// TwinCAT 3 PLC project AccelerationSensor
// ProgramVersion: 3.1.0.8
// libraries:
//   Tc2_SerialCom, * (Beckhoff Automation GmbH)
//   Tc2_Standard, * (Beckhoff Automation GmbH)
//   Tc2_Utilities, * (Beckhoff Automation GmbH)
//   Tc3_Module, * (Beckhoff Automation GmbH)
// project tree:
//   GVLs/ AccelerationSensor.TcGVL, ActivationStatus.TcDUT (not stored), DUT.TcDUT, GuidanceSystemSTM.TcDUT, GVL.TcGVL, HighLevelCondition.TcDUT (not stored), HLSInputData.TcDUT, HLSInputData_1.TcDUT, HLSInputs.TcDUT, HLSOutputs.TcDUT, LEDColor.TcDUT (not stored), LEDMode.TcDUT, LevitationSystemSTM.TcDUT, OperationControlCommands.TcDUT, ServiceModuleSTM.TcDUT, SubLevelCondition.TcDUT (not stored), TopLevelSTM.TcDUT
//   / PlcTask_Fast.TcTTO, PlcTask_Standard.TcTTO (not stored)
//   POUs/ FB_AccelerationSensor.TcPOU, FB_SerialComRS232.TcPOU, ITF_HighLevelSystem.TcIO, ITF_SubSystem.TcIO, MAIN.TcPOU
//   POUs/Mit Background/ Background.TcPOU (not stored), BackgroundEL.TcPOU, FB_SerialCom.TcPOU
// real-time tasks:
//   TASK PlcTask_Fast: cycle T#1ms, priority 19, ADS port 350
//   TASK PlcTask_Standard: cycle T#1ms, priority 20, ADS port 351
// I/O:
//   DEVICE Gerät 1 (EtherCAT), AmsNetId 10.183.66.136.2.1
//     Klemme 1 (EK1100) [EK1100 EtherCAT-Koppler (2A E-Bus)]
//       Klemme 2 (EL6001) [EL6001 Schnittstelle (RS232)]
//       Klemme 3 (EL9011) [EL9011 Endklemme]
// variable links:
//   AccelerationSensor/AccelerationSensor Instance <-> Device 1 (EtherCAT)/Term 1 (EK1100)/Term 2 (EL6001)
//     PlcTask_Standard Inputs/AccelerationSensor.stEL6001In @bit {16..184 step 8} <-> COM Inputs/Data In {0..21}  (22 links)
//     PlcTask_Standard Inputs/AccelerationSensor.stEL6001In <-> COM Inputs/Status
//     PlcTask_Standard Outputs/AccelerationSensor.stEL6001Out <-> COM Outputs/Ctrl
//     PlcTask_Standard Outputs/AccelerationSensor.stEL6001Out @bit {16..184 step 8} <-> COM Outputs/Data Out {0..21}  (22 links)

CONFIGURATION AccelerationSensor
    RESOURCE PLC ON TwinCAT3
        TASK PlcTask_Fast(INTERVAL := T#1ms, PRIORITY := 19);
        PROGRAM Background WITH PlcTask_Fast : Background;
    END_RESOURCE
END_CONFIGURATION

// ---- GVLs/DUT.TcDUT
TYPE DUT :
STRUCT
	b : BOOL;
	n : BOOL;
	m : BOOL;
END_STRUCT
END_TYPE

// ---- GVLs/GuidanceSystemSTM.TcDUT
{attribute 'qualified_only'}
{attribute 'strict'}
TYPE GuidanceSystemSTM :
(
	Idling,
	Initialising,
	PreRunning,
	Running,
	PostRunning
);
END_TYPE

// ---- GVLs/HLSInputData.TcDUT
TYPE HLSInputData :
STRUCT
	//In
	iIn : INT;
END_STRUCT
END_TYPE

// ---- GVLs/HLSInputData_1.TcDUT
TYPE HLSInputData_1 :
STRUCT
	//In
	iIn : INT;
	
	//Out
	iOut : INT;
END_STRUCT
END_TYPE

// ---- GVLs/HLSInputs.TcDUT
TYPE HLSInputs :
STRUCT
	iIn : INT;
END_STRUCT
END_TYPE

// ---- GVLs/HLSOutputs.TcDUT
TYPE HLSOutputs :
STRUCT
	iOut : INT;
END_STRUCT
END_TYPE

// ---- GVLs/LEDMode.TcDUT
{attribute 'qualified_only'}
{attribute 'strict'}
TYPE LEDMode :
(
	Off,
	On,
	Dimmed,
	SlowFlashing,
	FastFlashing
);
END_TYPE

// ---- GVLs/LevitationSystemSTM.TcDUT
{attribute 'qualified_only'}
{attribute 'strict'}
TYPE LevitationSystemSTM :
(
	Idling,
	Stationary,
	Transitioning,
	HoldingAirGap,
	TransitioningToZero
);
END_TYPE

// ---- GVLs/OperationControlCommands.TcDUT
TYPE OperationControlCommands :
STRUCT
	bStartOperational : BOOL;
	bStopOperational : BOOL;
	bGoToError : BOOL;
	bAckError : BOOL;
	nOperationMode : BYTE;
END_STRUCT
END_TYPE

// ---- GVLs/ServiceModuleSTM.TcDUT
{attribute 'qualified_only'}
{attribute 'strict'}
TYPE ServiceModuleSTM :
(
	Idling,
	Waiting,
	Running,
	PostRunning,
	PreparingForError
);
END_TYPE

// ---- GVLs/TopLevelSTM.TcDUT
{attribute 'qualified_only'}
{attribute 'strict'}
TYPE TopLevelSTM :
(
	STARTUP,
	READY,
	OPERATIONAL,
	SHUTDOWN,
	ERROR
)USINT;
END_TYPE

// ---- GVLs/AccelerationSensor.TcGVL
VAR_GLOBAL
	stEL6001In AT %I*	: EL6inData22B;		//**To EL6021 Inputs**
	stEL6001Out AT %Q*	: EL6outData22B;	//**To EL6021 Outputs**
END_VAR

// ---- GVLs/GVL.TcGVL
VAR_GLOBAL
	RxBufferEL			: ComBuffer;	(* Receive data buffer; used with all receive function blocks *)
	TxBufferEL			: ComBuffer;	(* Transmit data buffer; used with all receive function blocks *)
END_VAR

// ---- POUs/ITF_HighLevelSystem.TcIO
INTERFACE ITF_HighLevelSystem

PROPERTY eActivationStatus : ActivationStatus
GET
END_GET
SET
END_SET
END_PROPERTY

PROPERTY PUBLIC eCondition : HighLevelCondition
GET
END_GET
END_PROPERTY

PROPERTY PUBLIC nErrorID : UDINT
GET
END_GET
END_PROPERTY

END_INTERFACE

// ---- POUs/ITF_SubSystem.TcIO
INTERFACE ITF_SubSystem

PROPERTY PUBLIC eCondition : SubLevelCondition
GET
END_GET
END_PROPERTY

PROPERTY PUBLIC nErrorID : UDINT
GET
END_GET
END_PROPERTY

END_INTERFACE

// ---- POUs/FB_AccelerationSensor.TcPOU
FUNCTION_BLOCK FB_AccelerationSensor IMPLEMENTS ITF_SubSystem
VAR_OUTPUT
	aAccelerationValues : ARRAY [0..2] OF REAL;
END_VAR
VAR
	//Local
	fbEL6001	: FB_SerialComRS232;
	fPacketRate : REAL := 0;
	bStartPacketCount : BOOL;
	
	fbTimer : TON;
	fbReset : TON;
	fbTrigger : R_TRIG;
	nCounter1 : UDINT;
	nCounter2 : UDINT;
	aPackets : ARRAY [0..9] OF UDINT;
	i : UDINT := 0;
	nSum : UDINT := 0;
	bTrigger : BOOL := FALSE;
	
	//ErrorBits
	bCommunicationError : BIT;
	bOutOfRange : BIT;
END_VAR
VAR CONSTANT
	fGravitationalAcceleration : REAL := 9.81;  					//in m/s^2
END_VAR

fbEL6001(stEL6001In:=AccelerationSensor.stEL6001In, stEL6001Out:=AccelerationSensor.stEL6001Out);

aAccelerationValues := fbEL6001.aAcceleration;

doPacketCount();

METHOD PRIVATE doCheckRange : BOOL
VAR_INPUT
	aValues : ARRAY [0..2] OF REAL;
	fMax : REAL;
END_VAR
IF ABS(aValues[0]) <= fMax AND ABS(aValues[1]) <= fMax AND ABS(aValues[2]) <= fMax THEN
	doCheckRange := TRUE;
ELSE
	doCheckRange := FALSE;
END_IF
END_METHOD

METHOD PRIVATE doPacketCount
VAR_INPUT
END_VAR
fbTimer(IN := bStartPacketCount, PT := T#1S);
fbTrigger(CLK := fbTimer.IN);

IF fbTrigger.Q THEN
	nCounter1 := fbEL6001.nReceiveCounter;
END_IF

IF fbTimer.Q THEN
	nCounter2 := fbEL6001.nReceiveCounter;
	aPackets[i] := nCounter2 - nCounter1;
	nSum := nSum + aPackets[i];
	i := i + 1;
	bTrigger := TRUE;
	bStartPacketCount := FALSE;
END_IF

IF i = 10 THEN
	bTrigger := FALSE;
	fPacketRate := (UDINT_TO_REAL(nSum) / UDINT_TO_REAL(i));
	i := 0;
	nSum := 0;
END_IF

fbReset(IN := bTrigger, PT := T#3S);
IF fbReset.Q THEN
	bStartPacketCount := TRUE;
	bTrigger := FALSE;
END_IF
END_METHOD

PROPERTY PUBLIC eCondition : SubLevelCondition
GET
IF nErrorID <> 0 THEN
	eCondition := SubLevelCondition.ERROR;
ELSE
	eCondition := SubLevelCondition.RUN;
END_IF
END_GET
END_PROPERTY

PROPERTY PUBLIC nErrorID : UDINT
GET
IF fbEL6001.eReceiveErrorID <> COMERROR_NOERROR THEN
	bCommunicationError := TRUE;
ELSE
	bCommunicationError := FALSE;
END_IF

bOutOfRange := NOT doCheckRange(aValues:=aAccelerationValues, fMax:=2*fGravitationalAcceleration);


nErrorID.0 := bCommunicationError;
nErrorID.1 := bOutOfRange;
END_GET
END_PROPERTY

END_FUNCTION_BLOCK

// ---- POUs/FB_SerialComRS232.TcPOU
FUNCTION_BLOCK FB_SerialComRS232
VAR_IN_OUT

	stEL6001In : EL6inData22B;
	stEL6001Out : EL6outData22B;
END_VAR
VAR_OUTPUT
	aAcceleration : ARRAY [0..2] OF REAL;
	eReceiveErrorID	: ComError_t;
	nReceiveCounter	: UDINT;
END_VAR
VAR

	//Receive Buffer
	fbEL6001Ctrl		: SerialLineControl;
	TxBuffer	: ComBuffer;
	RxBuffer	: ComBuffer;
	//Receive Data
	fbReceive		: ReceiveData;
	nPrefix : ARRAY[0..1] OF BYTE;
	aReceiveData : ARRAY [0..15] OF BYTE;
	nPacketID : BYTE := 37;
	nPacketLength : BYTE := 12;	
	
	nCRC : WORD;
	nCheckCRC : WORD;
	nPointerCRC : POINTER TO WORD;
	aCRC : ARRAY [0..1] OF BYTE;	
	aDataArray : ARRAY[0..11] OF BYTE;
	i : USINT;
	aAccX : ARRAY [0..3] OF BYTE;
	aAccY : ARRAY [0..3] OF BYTE;
	aAccZ : ARRAY [0..3] OF BYTE;
	fPointerToX : POINTER TO REAL;
    fAccX : REAL;
	fPointerToY : POINTER TO REAL;
    fAccY : REAL;
	fPointerToZ : POINTER TO REAL;
    fAccZ : REAL;
END_VAR

fbEL6001Ctrl(
	Mode:= SERIALLINEMODE_EL6_22B, 
	pComIn:= ADR(stEL6001In), 
	pComOut:= ADR(stEL6001Out), 
	SizeComIn:= SIZEOF(stEL6001In), 
	Error=> , 
	ErrorID=> , 
	TxBuffer:= TxBuffer, 
	RxBuffer:= RxBuffer);

nPrefix[0] := nPacketID;
nPrefix[1] := nPacketLength;

fbReceive(
	RXbuffer:= RxBuffer,
	pPrefix := ADR(nPrefix),
	LenPrefix := 2,
	pReceiveData := ADR(aReceiveData),
	SizeReceiveData  := 16,								
	Error => eReceiveErrorID,
	DataReceived=>);
		
IF fbReceive.DataReceived THEN							
	nReceiveCounter := nReceiveCounter + 1;
END_IF

doCRC16Check();
doCalculateAccValues();

METHOD PRIVATE doCalculateAccValues
VAR_INPUT
END_VAR
IF nCheckCRC = nCRC THEN
	aAccX[0] := aReceiveData[4];
	aAccX[1] := aReceiveData[5];
	aAccX[2] := aReceiveData[6];
	aAccX[3] := aReceiveData[7];
	fPointerToX := ADR(aAccX);
	fAccX := fPointerToX^;
	
	aAccY[0] := aReceiveData[8];
	aAccY[1] := aReceiveData[9];
	aAccY[2] := aReceiveData[10];
	aAccY[3] := aReceiveData[11];
	fPointerToY := ADR(aAccY);
	fAccY := fPointerToY^;
	
	aAccZ[0] := aReceiveData[12];
	aAccZ[1] := aReceiveData[13];
	aAccZ[2] := aReceiveData[14];
	aAccZ[3] := aReceiveData[15];
	fPointerToZ := ADR(aAccZ);
	fAccZ := fPointerToZ^;
END_IF

aAcceleration[0] := fAccX;
aAcceleration[1] := fAccY;
aAcceleration[2] := fAccZ;
END_METHOD

METHOD PRIVATE doCRC16Check : BOOL
VAR_INPUT
END_VAR
FOR i:=0 TO 11 DO
	aDataArray[i] := aReceiveData[i+4];
END_FOR


nCRC := F_DATA_TO_CRC16_CCITT(
	pData := ADR(aDataArray),
	cbData := BYTE_TO_UDINT(nPacketLength),
	crc := 16#FFFF);

aCRC[0] := aReceiveData[2];
aCRC[1] := aReceiveData[3];
nPointerCRC := ADR(aCRC);
nCheckCRC := nPointerCRC^;
END_METHOD

END_FUNCTION_BLOCK

// ---- POUs/MAIN.TcPOU
PROGRAM MAIN
VAR
	fbIMU : FB_AccelerationSensor;
	
	x : REAL;
	y : REAL;
	z : REAL;
	
	acc : ARRAY [0..2] OF REAL;

//	fbEL6001	: FB_SerialCom;
	
//	(* exchange buffers with background communication with the PC COM port device *)
//	RxBufferPcCom	: ComBuffer;	(* Receive data buffer; used with all receive function blocks *)
//	TxBufferPcCom	: ComBuffer;	(* Transmit data buffer; used with all receive function blocks *)
	
//	acc_x : REAL;
//	acc_y : REAL;	
//	acc_z : REAL;
////	acc_x2 : REAL;
////	acc_y2 : REAL;	
////	acc_z2 : REAL;
////	acc_x3 : REAL;
////	acc_y3 : REAL;	
////	acc_z3 : REAL;
////	acc_x4 : REAL;
////	acc_y4 : REAL;	
////	acc_z4 : REAL;

//	fbTimer : TON;
//	fbReset : TON;
//	fbTrigger : R_TRIG;
//	iCounter1 : UDINT;
//	iCounter2 : UDINT;
//	a_iPackets : ARRAY [0..9] OF UDINT;
//	i : UDINT := 0;
//	iSum : UDINT := 0;
//	rPacketRate : REAL := 0;
//	bTrigger : BOOL := FALSE;
//	bCount : BOOL;

END_VAR

fbIMU();

acc := fbIMU.aAccelerationValues;

x := acc[0];
y := acc[1];
z := acc[2];



//fbEL6001(TxBuffer:=TxBufferEL, RxBuffer:=RxBufferEL);

//acc_x := fbEL6001.getAccelerationValueX;
//acc_y := fbEL6001.getAccelerationValueY;
//acc_z := fbEL6001.getAccelerationValueZ;

//acc_x2 := fbEL6001.getAccelerationValueX2;
//acc_y2 := fbEL6001.getAccelerationValueY2;
//acc_z2 := fbEL6001.getAccelerationValueZ2;

//acc_x3 := fbEL6001.getAccelerationValueX3;
//acc_y3 := fbEL6001.getAccelerationValueY3;
//acc_z3 := fbEL6001.getAccelerationValueZ3;

//acc_x4 := fbEL6001.getAccelerationValueX4;
//acc_y4 := fbEL6001.getAccelerationValueY4;
//acc_z4 := fbEL6001.getAccelerationValueZ4;

doPacketCount();					//start packet count by setting bCount 'true' --> rPacketRate shows average rate per second

METHOD doPacketCount : REAL
VAR_INPUT
END_VAR
//fbTimer(IN := bCount, PT := T#1S);
//fbTrigger(CLK := fbTimer.IN);

//IF fbTrigger.Q THEN
//	iCounter1 := fbEL6001.nReceiveCounter;
//END_IF

//IF fbTimer.Q THEN
//	iCounter2 := fbEL6001.nReceiveCounter;
//	a_iPackets[i] := iCounter2 - iCounter1;
//	iSum := iSum + a_iPackets[i];
//	i := i + 1;
//	bTrigger := TRUE;
//	bCount := FALSE;
//END_IF

//IF i = 10 THEN
//	bTrigger := FALSE;
//	rPacketRate := (UDINT_TO_REAL(iSum) / UDINT_TO_REAL(i));			//times amount of packets
//	i := 0;
//	iSum := 0;
//END_IF

//fbReset(IN := bTrigger, PT := T#3S);
//IF fbReset.Q THEN
//	bCount := TRUE;
//	bTrigger := FALSE;
//END_IF
END_METHOD

END_PROGRAM

// ---- POUs/Mit Background/BackgroundEL.TcPOU
PROGRAM BackgroundEL
VAR
	(* background communication with the EL6001 terminal *)
	fbEL6001Ctrl		: SerialLineControl;
	bEL6001CtrlError	: BOOL;
	eEL6001CtrlErrorID	: ComError_t;
	(* 	I/O variables for a EL6001 terminal*)
	stIn_EL6001 AT %I*	: EL6inData22B;	(* linked to the EL6001 in the TwinCAT System Manager *)
	stOut_EL6001 AT %Q*	: EL6outData22B;(* linked to the EL6001 in the TwinCAT System Manager *)
END_VAR

fbEL6001Ctrl(
	Mode:= SERIALLINEMODE_EL6_22B, 
	pComIn:= ADR(stIn_EL6001), 
	pComOut:= ADR(stOut_EL6001), 
	SizeComIn:= SIZEOF(stIn_EL6001), 
	Error=> , 
	ErrorID=> , 
	TxBuffer:= TxBufferEL, 
	RxBuffer:= RxBufferEL );
IF fbEL6001Ctrl.Error THEN
	bEL6001CtrlError := TRUE;
	eEL6001CtrlErrorID := fbEL6001Ctrl.ErrorID;
END_IF

END_PROGRAM

// ---- POUs/Mit Background/FB_SerialCom.TcPOU
FUNCTION_BLOCK FB_SerialCom
VAR_IN_OUT
	TxBuffer	: ComBuffer;
	RxBuffer	: ComBuffer;
END_VAR
VAR
	fbReceive		: ReceiveData;
	eReceiveErrorID	: ComError_t;
	nReceiveCounter	: UDINT;
	prefix : ARRAY[0..1] OF BYTE;
	receivedata : ARRAY [0..15] OF BYTE;					//decrease or increase by 17 pro packet
	packet_ID : BYTE := 37;
	packet_length : BYTE := 12;	
	
	//First Package
	crc : WORD;
	crc_check : WORD;
	pt_crc : POINTER TO WORD;
	crc12 : ARRAY [0..1] OF BYTE;	
	dataArray : ARRAY[0..11] OF BYTE;
	i : USINT;
	acc_x : ARRAY [0..3] OF BYTE;
	acc_y : ARRAY [0..3] OF BYTE;
	acc_z : ARRAY [0..3] OF BYTE;
	pt_x : POINTER TO REAL;
    x_acc : REAL;
	pt_y : POINTER TO REAL;
    y_acc : REAL;
	pt_z : POINTER TO REAL;
    z_acc : REAL;
	

//	//Second Package
//	bSecondReceivedData: ARRAY [0..16] OF BYTE;
//	dataArray2 : ARRAY[0..11] OF BYTE;
//	crc2 : WORD;
//	crc122 : ARRAY [0..1]OF BYTE;
//	pt_crc2 : POINTER TO WORD;
//	crc_check2 : WORD;
//	k2 : USINT;
//	LRCsum2 : BYTE;
//	LRC2 : BYTE;
//	LRCchecked2 : BOOL;
//	j2 : USINT;
//	bIn2 : BOOL;
//	acc_x2 : ARRAY [0..3] OF BYTE;
//	acc_y2 : ARRAY [0..3] OF BYTE;
//	acc_z2 : ARRAY [0..3] OF BYTE;
//	pt_x2 : POINTER TO REAL;
//  x_acc2 : REAL;
//	pt_y2 : POINTER TO REAL;
//  y_acc2 : REAL;
//	pt_z2 : POINTER TO REAL;
//  z_acc2 : REAL;
	
//	//Third Package
//	bThirdReceivedData: ARRAY [0..16] OF BYTE;
//	dataArray3 : ARRAY[0..11] OF BYTE;
//	crc3 : WORD;
//	crc123 : ARRAY [0..1]OF BYTE;
//	pt_crc3 : POINTER TO WORD;
//	crc_check3 : WORD;
//	k3 : USINT;
//	LRCsum3 : BYTE;
//	LRC3 : BYTE;
//	LRCchecked3 : BOOL;
//	j3 : USINT;
//	bIn3 : BOOL;
//	acc_x3 : ARRAY [0..3] OF BYTE;
//	acc_y3 : ARRAY [0..3] OF BYTE;
//	acc_z3 : ARRAY [0..3] OF BYTE;
//	pt_x3 : POINTER TO REAL;
//  x_acc3 : REAL;
//	pt_y3 : POINTER TO REAL;
//  y_acc3 : REAL;
//	pt_z3 : POINTER TO REAL;
//  z_acc3 : REAL;
	
//	//Fourth Package
//	bFourthReceivedData: ARRAY [0..16] OF BYTE;
//	dataArray4 : ARRAY[0..11] OF BYTE;
//	crc4 : WORD;
//	crc124 : ARRAY [0..1]OF BYTE;
//	pt_crc4 : POINTER TO WORD;
//	crc_check4 : WORD;
//	k4 : USINT;
//	LRCsum4 : BYTE;
//	LRC4 : BYTE;
//	LRCchecked4 : BOOL;
//	j4 : USINT;
//	bIn4 : BOOL;
//	acc_x4 : ARRAY [0..3] OF BYTE;
//	acc_y4 : ARRAY [0..3] OF BYTE;
//	acc_z4 : ARRAY [0..3] OF BYTE;
//	pt_x4 : POINTER TO REAL;
//  x_acc4 : REAL;
//	pt_y4 : POINTER TO REAL;
//  y_acc4 : REAL;
//	pt_z4 : POINTER TO REAL;
//  z_acc4 : REAL;
END_VAR

prefix[0] := packet_ID;
prefix[1] := packet_length;

fbReceive(
	RXbuffer:= RxBuffer,
	pPrefix := ADR(prefix),
	LenPrefix := 2,
	pReceiveData := ADR(receivedata),
	SizeReceiveData  := 16,											//decrease or increase by 17 per packet
	Error=> ,
	DataReceived=>,
		);
IF fbReceive.Error <> COMERROR_NOERROR THEN
	eReceiveErrorID := fbReceive.Error;
END_IF
IF fbReceive.DataReceived THEN										//check bIn* variables as well for multiple packets
	nReceiveCounter := nReceiveCounter + 1;
END_IF

doCRC16Check1();

//IF receivedata[17] = 37 AND receivedata[18] = 12 THEN				//decrease or increase by 17 per packet
//	bIn2 := TRUE;	
//	FOR k2:=0 TO 16 DO
//		bSecondReceivedData[k] := receivedata[k+16];
//	END_FOR
	
//	doLRCCheck2();
//	doCRC16Check2();
//ELSE
//	bIn2 := FALSE;
//END_IF


//IF receivedata[34] = 37 AND receivedata[35] = 12 THEN				//decrease or increase by 17 per packet
//	bIn3 := TRUE;	
//	FOR k3:=0 TO 16 DO
//		bThirdReceivedData[k3] := receivedata[k3+16];
//	END_FOR
	
//	doLRCCheck3();
//	doCRC16Check3();
//ELSE
//	bIn3 := FALSE;
//END_IF


//IF receivedata[51] = 37 AND receivedata[52] = 12 THEN			//decrease or increase by 17 per packet
//	bIn4 := TRUE;	
//	FOR k4:=0 TO 16 DO
//		bFourthReceivedData[k4] := receivedata[k4+16];
//	END_FOR
	
//	doLRCCheck4();
//	doCRC16Check4();
//ELSE
//	bIn4 := FALSE;
//END_IF

METHOD doCRC16Check1 : BOOL
VAR_INPUT
END_VAR
FOR i:=0 TO 11 DO
	dataArray[i] := receivedata[i+4];
END_FOR


crc := F_DATA_TO_CRC16_CCITT(
	pData := ADR(dataArray),
	cbData := BYTE_TO_UDINT(packet_length),
	crc := 16#FFFF);

crc12[0] := receivedata[2];
crc12[1] := receivedata[3];
pt_crc := ADR(crc12);
crc_check := pt_crc^;
END_METHOD

METHOD doCRC16Check2 : BOOL
VAR_INPUT
END_VAR
//FOR j2:=0 TO 11 DO
//	dataArray2[j] := bSecondReceivedData[j+5];
//END_FOR
	
	
//crc2 := F_DATA_TO_CRC16_CCITT(
//	pData := ADR(dataArray2),
//	cbData := BYTE_TO_UDINT(packet_length),
//	crc := 16#FFFF);

//crc122[0] := bSecondReceivedData[3];
//crc122[1] := bSecondReceivedData[4];
//pt_crc2 := ADR(crc122);
//crc_check2 := pt_crc2^;
END_METHOD

METHOD doCRC16Check3 : BOOL
VAR_INPUT
END_VAR
//FOR j3:=0 TO 11 DO
//	dataArray3[j3] := bThirdReceivedData[j3+5];
//END_FOR
	
	
//crc3 := F_DATA_TO_CRC16_CCITT(
//	pData := ADR(dataArray3),
//	cbData := BYTE_TO_UDINT(packet_length),
//	crc := 16#FFFF);

//crc123[0] := bThirdReceivedData[3];
//crc123[1] := bThirdReceivedData[4];
//pt_crc3 := ADR(crc123);
//crc_check3 := pt_crc3^;
END_METHOD

METHOD doCRC16Check4 : BOOL
VAR_INPUT
END_VAR
//FOR j4:=0 TO 11 DO
//	dataArray4[j4] := bFourthReceivedData[j4+5];
//END_FOR
	
	
//crc4 := F_DATA_TO_CRC16_CCITT(
//	pData := ADR(dataArray4),
//	cbData := BYTE_TO_UDINT(packet_length),
//	crc := 16#FFFF);

//crc124[0] := bFourthReceivedData[3];
//crc124[1] := bFourthReceivedData[4];
//pt_crc4 := ADR(crc124);
//crc_check4 := pt_crc4^;
END_METHOD

METHOD doLRCCheck2 : BOOL
VAR_INPUT
END_VAR
//LRCsum2 := (bSecondReceivedData[1] + bSecondReceivedData[2] + bSecondReceivedData[3] + bSecondReceivedData[4]) XOR 255;
//LRC2 := bSecondReceivedData[0] - 1;
//LRCchecked2 := (LRCsum2 = LRC2);
END_METHOD

METHOD doLRCCheck3 : BOOL
VAR_INPUT
END_VAR
//LRCsum3 := (bThirdReceivedData[1] + bThirdReceivedData[2] + bThirdReceivedData[3] + bThirdReceivedData[4]) XOR 255;
//LRC3 := bThirdReceivedData[0] - 1;
//LRCchecked3 := (LRCsum3 = LRC3);
END_METHOD

METHOD doLRCCheck4 : BOOL
VAR_INPUT
END_VAR
//LRCsum4 := (bFourthReceivedData[1] + bFourthReceivedData[2] + bFourthReceivedData[3] + bFourthReceivedData[4]) XOR 255;
//LRC4 := bFourthReceivedData[0] - 1;
//LRCchecked4 := (LRCsum4 = LRC4);
END_METHOD

PROPERTY getAccelerationValueX : REAL
GET
IF crc_check = crc THEN

	acc_x[0] := receivedata[4];
	acc_x[1] := receivedata[5];
	acc_x[2] := receivedata[6];
	acc_x[3] := receivedata[7];
	pt_x := ADR(acc_x);
	x_acc := pt_x^;
END_IF

getAccelerationValueX := x_acc;
END_GET
END_PROPERTY

PROPERTY getAccelerationValueX2 : REAL
GET
//IF LRCsum = LRC AND crc2 = crc_check2 THEN
//	acc_x2[0] := bSecondReceivedData[5];
//	acc_x2[1] := bSecondReceivedData[6];
//	acc_x2[2] := bSecondReceivedData[7];
//	acc_x2[3] := bSecondReceivedData[8];
//	pt_x2 := ADR(acc_x2);
//	x_acc2 := pt_x2^;
//END_IF

//getAccelerationValueX2 := x_acc2;
END_GET
END_PROPERTY

PROPERTY getAccelerationValueX3 : REAL
GET
//IF LRCsum3 = LRC3 AND crc3 = crc_check3 THEN
//	acc_x3[0] := bThirdReceivedData[5];
//	acc_x3[1] := bThirdReceivedData[6];
//	acc_x3[2] := bThirdReceivedData[7];
//	acc_x3[3] := bThirdReceivedData[8];
//	pt_x3 := ADR(acc_x3);
//	x_acc3 := pt_x3^;
//END_IF

//getAccelerationValueX3 := x_acc3;
END_GET
END_PROPERTY

PROPERTY getAccelerationValueX4 : REAL
GET
//IF LRCsum4 = LRC4 AND crc4 = crc_check4 THEN
//	acc_x4[0] := bFourthReceivedData[5];
//	acc_x4[1] := bFourthReceivedData[6];
//	acc_x4[2] := bFourthReceivedData[7];
//	acc_x4[3] := bFourthReceivedData[8];
//	pt_x4 := ADR(acc_x4);
//	x_acc4 := pt_x4^;
//END_IF

//getAccelerationValueX4 := x_acc4;
END_GET
END_PROPERTY

PROPERTY getAccelerationValueY : REAL
GET
IF crc_check = crc THEN
	
	acc_y[0] := receivedata[8];
	acc_y[1] := receivedata[9];
	acc_y[2] := receivedata[10];
	acc_y[3] := receivedata[11];
	pt_y := ADR(acc_y);
	y_acc := pt_y^;

END_IF
getAccelerationValueY := y_acc;
END_GET
END_PROPERTY

PROPERTY getAccelerationValueY2 : REAL
GET
//IF LRCsum = LRC AND crc2 = crc_check2 THEN
//	acc_y2[0] := bSecondReceivedData[9];
//	acc_y2[1] := bSecondReceivedData[10];
//	acc_y2[2] := bSecondReceivedData[11];
//	acc_y2[3] := bSecondReceivedData[12];
//	pt_y2 := ADR(acc_y2);
//	y_acc2 := pt_y2^;
//END_IF

//getAccelerationValueY2 := y_acc2;
END_GET
END_PROPERTY

PROPERTY getAccelerationValueY3 : REAL
GET
//IF LRCsum3 = LRC3 AND crc3 = crc_check3 THEN
//	acc_y3[0] := bThirdReceivedData[9];
//	acc_y3[1] := bThirdReceivedData[10];
//	acc_y3[2] := bThirdReceivedData[11];
//	acc_y3[3] := bThirdReceivedData[12];
//	pt_y3 := ADR(acc_y3);
//	y_acc3 := pt_y3^;
//END_IF

//getAccelerationValueY3 := y_acc3;
END_GET
END_PROPERTY

PROPERTY getAccelerationValueY4 : REAL
GET
//IF LRCsum4 = LRC4 AND crc4 = crc_check4 THEN
//	acc_y4[0] := bFourthReceivedData[9];
//	acc_y4[1] := bFourthReceivedData[10];
//	acc_y4[2] := bFourthReceivedData[11];
//	acc_y4[3] := bFourthReceivedData[12];
//	pt_y4 := ADR(acc_y4);
//	y_acc4 := pt_y4^;
//END_IF

//getAccelerationValueY4 := y_acc4;
END_GET
END_PROPERTY

PROPERTY getAccelerationValueZ : REAL
GET
IF crc_check = crc THEN
	
	acc_z[0] := receivedata[12];
	acc_z[1] := receivedata[13];
	acc_z[2] := receivedata[14];
	acc_z[3] := receivedata[15];
	pt_z := ADR(acc_z);
	z_acc := pt_z^;
END_IF

getAccelerationValueZ := z_acc;
END_GET
END_PROPERTY

PROPERTY getAccelerationValueZ2 : REAL
GET
//IF LRCsum = LRC AND crc2 = crc_check2 THEN
//	acc_z2[0] := bSecondReceivedData[13];
//	acc_z2[1] := bSecondReceivedData[14];
//	acc_z2[2] := bSecondReceivedData[15];
//	acc_z2[3] := bSecondReceivedData[16];
//	pt_z2 := ADR(acc_z2);
//	z_acc2 := pt_z2^;
//END_IF

//getAccelerationValueZ2 := z_acc2;
END_GET
END_PROPERTY

PROPERTY getAccelerationValueZ3 : REAL
GET
//IF LRCsum3 = LRC3 AND crc3 = crc_check3 THEN
//	acc_z3[0] := bThirdReceivedData[13];
//	acc_z3[1] := bThirdReceivedData[14];
//	acc_z3[2] := bThirdReceivedData[15];
//	acc_z3[3] := bThirdReceivedData[16];
//	pt_z3 := ADR(acc_z3);
//	z_acc3 := pt_z3^;
//END_IF

//getAccelerationValueZ3 := z_acc3;
END_GET
END_PROPERTY

PROPERTY getAccelerationValueZ4 : REAL
GET
//IF LRCsum4 = LRC4 AND crc4 = crc_check4 THEN
//	acc_z4[0] := bFourthReceivedData[13];
//	acc_z4[1] := bFourthReceivedData[14];
//	acc_z4[2] := bFourthReceivedData[15];
//	acc_z4[3] := bFourthReceivedData[16];
//	pt_z4 := ADR(acc_z4);
//	z_acc4 := pt_z4^;
//END_IF

//getAccelerationValueZ4 := z_acc4;
END_GET
END_PROPERTY

END_FUNCTION_BLOCK
